// TIA Portal V17 export
// export: Created 2024-06-16T17:47:24.4798873Z, ExportSetting WithDefaults, DisplayName Totally Integrated Automation Portal, DisplayVersion V17, DisplayName TIA Portal Openness, DisplayVersion V17, DisplayName TIA Portal Version Control Interface, DisplayVersion V17, DisplayName STEP 7 Professional, DisplayVersion V17, DisplayName STEP 7 Safety, DisplayVersion V17, DisplayName WinCC Professional, DisplayVersion V17
DATA_BLOCK "Cfg_St1_Prehenseur_Z"   // DB180
AUTHOR : DRVDPS7
FAMILY : DRIVES
NAME : SINA_POS
VERSION : 5.7
// stored: AutoNumber false, DBAccessibleFromOPCUA true, DBAccessibleFromWebserver true, InstanceOfName SINA_POS, InstanceOfType FB
"SINA_POS"
   // VAR_INPUT
   //    ModePos : Int;
   //    EnableAxis : Bool;
   //    CancelTraversing : Bool;
   //    IntermediateStop : Bool;
   //    Positive : Bool;
   //    Negative : Bool;
   //    Jog1 : Bool;
   //    Jog2 : Bool;
   //    FlyRef : Bool;
   //    AckError : Bool;
   //    ExecuteMode : Bool;
   //    Position : DInt;
   //    Velocity : DInt;
   //    OverV : Int;
   //    OverAcc : Int;
   //    OverDec : Int;
   //    ConfigEPos : DWord;
   //    HWIDSTW : HW_IO;
   //    HWIDZSW : HW_IO;
   // END_VAR
   // VAR_OUTPUT
   //    AxisEnabled : Bool;
   //    AxisPosOk : Bool;
   //    AxisSpFixed : Bool;
   //    AxisRef : Bool;
   //    AxisWarn : Bool;
   //    AxisError : Bool;
   //    Lockout : Bool;
   //    ActVelocity : DInt;
   //    ActPosition : DInt;
   //    ActMode : Int;
   //    EPosZSW1 : Word;
   //    EPosZSW2 : Word;
   //    ActWarn : Word;
   //    ActFault : Word;
   //    Error : Bool;
   //    Status : Word;
   //    DiagID : Word;
   // END_VAR
   // VAR
   //    sbOff1Edge : Bool;
   //    sbOff1 : Bool;
   //    sbExecuteEdge : Bool;
   //    sbExecute : Bool;
   //    sbRefTypEdge : Bool;
   //    sbRefTyp : Bool;
   //    sbMdiStart : Bool;
   //    sbMdiStartEdge : Bool;
   //    sbRefStart : Bool;
   //    sbJogInc : Bool;
   //    sbReady : Bool;
   //    sbIOp : Bool;
   //    sbAccel : Bool;
   //    sbDecel : Bool;
   //    sbAlarm : Bool;
   //    sbFault : Bool;
   //    sbFWD : Bool;
   //    sbBWD : Bool;
   //    sbBusy : Bool;
   //    swStatus : Word;
   //    swEPosZSW1 : Word;
   //    swEPosZSW2 : Word;
   //    siExecuteCyc : Int;
   //    siRefTypCyc : Int;
   //    siJogIncCyc : Int;
   //    siMdiStartCyc : Int;
   //    siRefActRetry : Int;
   //    siModePos : Int;
   //    siModePosMax : Int;
   //    siCycWait : Int;
   //    siRetryMax : Int;
   //    sbModePos : Bool;
   //    sxSendBuf : Struct
   //       STW1 : Word;
   //       EPosSTW1 : Word;
   //       EPosSTW2 : Word;
   //       STW2 : Word;
   //       OverrideV : Word;
   //       Position : DWord;
   //       Velocity : DWord;
   //       OverrideA : Word;
   //       OverrideD : Word;
   //       Reserve : Word;
   //    END_STRUCT;
   //    sxRecvBuf : Struct
   //       ZSW1 : Word;
   //       EPosZSW1 : Word;
   //       EPosZSW2 : Word;
   //       ZSW2 : Word;
   //       NotUsed : Word;
   //       Position : DWord;
   //       Velocity : DWord;
   //       ErrNr : Word;
   //       WarnNr : Word;
   //       Reserve : Word;
   //    END_STRUCT;
   // END_VAR
BEGIN
END_DATA_BLOCK
